PROGRAM MAIN
VAR
END_VAR

END_PROGRAM

(* stored: Version 1.1.0.1
   POU MAIN: Id {669211bc-d000-4e15-a5de-cc33797619a0} *)
